TYPE "MatCountData"
VERSION : 0.1
// Block: MatCountData
   STRUCT
      Standstill : Bool;
      CounterValid : Bool;
      AxPosition : LReal;
      AxPositionPrevious : LReal;
      FAK : LReal;
      CounterValueInit : LReal;
      CounterOffset : LReal;
      CounterValue : LReal;
      FAKPrevious : LReal;
      AX_MODULE : LReal;
      COUNTER_MODULE : LReal;
   END_STRUCT;

END_TYPE
